// TIA Portal V16 export
// export: Created 2022-04-01T14:07:08.3750457Z, ExportSetting WithDefaults, DisplayName Totally Integrated Automation Portal, DisplayVersion V16 Update 3, DisplayName TIA Portal Version Control Interface, DisplayVersion V16 Update 2, DisplayName TIA Portal Openness, DisplayVersion V16 Update 3, DisplayName STEP 7 Professional, DisplayVersion V16 Update 3, DisplayName STEP 7 Safety, DisplayVersion V16, DisplayName WinCC Professional, DisplayVersion V16 Update 3
TYPE "UT01001_St_SysLicence"
TITLE = Static UDT [SYSTEM] — Licence Information
// PRACTICAL SERIES AUTOMATION LIBRARY (PAL)   —   COPYRIGHT 2020 – M. GLEDHILL (MIT LICENCE)
//                   ———— ◆ ————
// FULL ONLINE DOCUMENTATION IS AVAILABLE AT: https://practicalseries.com/2001-pal/index.html
// stored: IsFailsafeCompliant false
   STRUCT
      LICENCE_TYPE { ExternalWritable := 'False'} : String[20];   // Licence information — type of licence
      COPYRIGHT { ExternalWritable := 'False'} : String[30];   // Licence information — copyright (year and name)
   END_STRUCT;
END_TYPE
